// TwinCAT 3 PLC project convey
// ProgramVersion: 3.1.0.9
// libraries:
//   VisuElem3DPath, 3.5.6.0 (System)
//   VisuElemMeter, 3.5.6.0 (System)
//   VisuElems, 3.5.6.10 (System)
//   VisuElemsDateTime, 3.5.6.0 (System)
//   VisuElemsSpecialControls, 3.5.6.0 (System)
//   VisuElemsWinControls, 3.5.6.0 (System)
//   VisuElemTextEditor, 3.5.6.0 (System)
//   visuinputs, 3.5.6.0 (system)
//   VisuNativeControl, 3.5.6.0 (System)
//   Tc2_Standard, * (Beckhoff Automation GmbH)
//   Tc2_System, * (Beckhoff Automation GmbH)
//   Tc3_Interfaces, * (Beckhoff Automation GmbH)
//   Tc3_Module, * (Beckhoff Automation GmbH)
//   VisuDialogs, * (System)
// project tree:
//   / Buttons.TcIPO (not stored), GlobalImagePool.TcGIPO (not stored), GlobalTextList.TcGTLO, ImagePool.TcIPO (not stored), PlcTask.TcTTO, stateImages.TcIPO (not stored), Visualization Manager.TcVMO (not stored), VISU_TASK.TcTTO
//   GVLs/ GVL.TcGVL
//   POUs/ autoMode.TcPOU, caseImageUpdate.TcPOU, leftBelt.TcPOU, leftLift.TcPOU, MAIN.TcPOU, manualMode.TcPOU, bottomBelt.TcPOU, readState.TcPOU, relaxPistons.TcPOU, rightBelt.TcPOU, rightLift.TcPOU, topBelt.TcPOU
//   VISUs/ about.TcVIS, allControls.TcVIS, autoMode.TcVIS, Main.TcVIS, manualMode.TcVIS
// real-time tasks:
//   TASK PlcTask: cycle T#10ms, priority 20, ADS port 350
//   TASK VISU_TASK: cycle T#100000us, priority 30, ADS port 351
// I/O:
//   DEVICE Device 1 (EtherCAT), AmsNetId 172.24.66.56.2.1
//     Term 1 (EK1100) [EK1100 EtherCAT Coupler (2A E-Bus)]
//       Term 2 (EL1008) [EL1008 8Ch. Dig. Input 24V, 3ms]
//       Term 3 (EL2008) [EL2008 8Ch. Dig. Output 24V, 0.5A]
//       Term 4 (EL3002) [EL3002 2Ch. Ana. Input +/-10V]
//       Term 5 (EL4002) [EL4002 2Ch. Ana. Output 0-10V, 12bit]
//       Term 6 (EL3124) [EL3124 4Ch. Ana. Input 4-20mA Diff.]
//       Term 7 (EL4024) [EL4024 4Ch. Ana. Output 4-20mA, 12bit]
//       Term 10 (EL9011) [EL9011 End Terminal]
//     Term 8 (EK1100) [EK1100 EtherCAT Coupler (2A E-Bus)]
//       Box 9 (BK1250)
//   DEVICE Device 2 (EtherCAT Automation Protocol), AmsNetId 172.24.66.56.3.1
// variable links:
//   convey/convey Instance <-> Device 1 (EtherCAT)/Term 8 (EK1100)/Box 9 (BK1250)
//     PlcTask Inputs/GVL.I_bInput11 <-> Term 4 (KL1104)/Channel 3/GVL.I_bInput11
//     PlcTask Inputs/GVL.I_bInput12 <-> Term 4 (KL1104)/Channel 4/GVL.I_bInput12
//     PlcTask Inputs/GVL.I_bLeftLiftBottom <-> Term 3 (KL1104)/Channel 2/GVL.I_bLeftLiftBottom
//     PlcTask Inputs/GVL.I_bLeftLiftUp <-> Term 3 (KL1104)/Channel 1/GVL.I_bLeftLiftUp
//     PlcTask Inputs/GVL.I_bLowBeltLeft <-> Term 4 (KL1104)/Channel 1/GVL.I_bLowBeltLeft
//     PlcTask Inputs/GVL.I_bLowBeltRight <-> Term 3 (KL1104)/Channel 3/GVL.I_bLowBeltRight
//     PlcTask Inputs/GVL.I_bPieceLeftLift <-> Term 2 (KL1104)/Channel 1/GVL.I_bPieceLeftLift
//     PlcTask Inputs/GVL.I_bPieceRightLift <-> Term 2 (KL1104)/Channel 2/GVL.I_bPieceRightLift
//     PlcTask Inputs/GVL.I_bRightLiftBottom <-> Term 2 (KL1104)/Channel 4/GVL.I_bRightLiftBottom
//     PlcTask Inputs/GVL.I_bRightLiftUp <-> Term 2 (KL1104)/Channel 3/GVL.I_bRightLiftUp
//     PlcTask Inputs/GVL.I_bTopBeltRight <-> Term 3 (KL1104)/Channel 4/GVL.I_bTopBeltRight
//     PlcTask Inputs/GVL.I_bTopBeltleft <-> Term 4 (KL1104)/Channel 2/GVL.I_bTopBeltleft
//     PlcTask Outputs/GVL.O_bLeftLiftBeltLeft <-> Term 6 (KL2114)/Channel 4/GVL.O_bLeftLiftBeltLeft
//     PlcTask Outputs/GVL.O_bLeftLiftBeltRight <-> Term 6 (KL2114)/Channel 3/GVL.O_bLeftLiftBeltRight
//     PlcTask Outputs/GVL.O_bLeftLiftDown <-> Term 5 (KL2114)/Channel 2/GVL.O_bLeftLiftDown
//     PlcTask Outputs/GVL.O_bLeftLiftUp <-> Term 5 (KL2114)/Channel 1/GVL.O_bLeftLiftUp
//     PlcTask Outputs/GVL.O_bLowBeltLeft <-> Term 7 (KL2114)/Channel 4/GVL.O_bLowBeltLeft
//     PlcTask Outputs/GVL.O_bLowBeltRight <-> Term 7 (KL2114)/Channel 2/GVL.O_bLowBeltRight
//     PlcTask Outputs/GVL.O_bRightLiftBeltLeft <-> Term 6 (KL2114)/Channel 1/GVL.O_bRightLiftBeltLeft
//     PlcTask Outputs/GVL.O_bRightLiftBeltRight <-> Term 6 (KL2114)/Channel 2/GVL.O_bRightLiftBeltRight
//     PlcTask Outputs/GVL.O_bRightLiftDown <-> Term 5 (KL2114)/Channel 3/GVL.O_bRightLiftDown
//     PlcTask Outputs/GVL.O_bRightLiftUp <-> Term 5 (KL2114)/Channel 4/GVL.O_bRightLiftUp
//     PlcTask Outputs/GVL.O_bTopBeltLeft <-> Term 7 (KL2114)/Channel 1/GVL.O_bTopBeltLeft
//     PlcTask Outputs/GVL.O_bTopBeltRight <-> Term 7 (KL2114)/Channel 3/GVL.O_bTopBeltRight

CONFIGURATION convey
    RESOURCE PLC ON TwinCAT3
        TASK PlcTask(INTERVAL := T#10ms, PRIORITY := 20);
        TASK VISU_TASK(INTERVAL := T#100000us, PRIORITY := 30);
        PROGRAM MAIN WITH PlcTask : MAIN;
        PROGRAM VisuElems_Visu_Prg WITH VISU_TASK : VisuElems.Visu_Prg;
    END_RESOURCE
END_CONFIGURATION

// ---- GVLs/GVL.TcGVL
VAR_GLOBAL
	I_bPieceLeftLift              AT %I*: BOOL; // DI 1 - Piece in the left lift
	I_bPieceRightLift             AT %I*: BOOL; // DI 2 - Piece in the right lift
	I_bRightLiftBottom            AT %I*: BOOL; // DI 3 - Right lift is bottom
	I_bRightLiftUp                AT %I*: BOOL; // DI 4 - Right lift is up
	I_bLeftLiftBottom             AT %I*: BOOL; // DI 5 - Left lift is down
	I_bLeftLiftUp                 AT %I*: BOOL; // DI 6 - Left lift is up
	I_bLowBeltRight 	          AT %I*: BOOL; // DI 7 - Piece on low belt right side
	I_bTopBeltRight               AT %I*: BOOL; // DI 8 - Piece on top belt right side
	I_bLowBeltLeft                AT %I*: BOOL; // DI 9 - Piece on low belt left side
	I_bTopBeltleft                AT %I*: BOOL; // DI 10 - Piece on top belt left side
	I_bInput11                    AT %I*: BOOL; // DI 11 - Empty
	I_bInput12                    AT %I*: BOOL; // DI 12 - Empty
	I_STARTbutton				  AT %I*: BOOL;
	
	O_bLeftLiftUp                 AT %Q*: BOOL; // DO 1 - Left Lift up
	O_bLeftLiftDown               AT %Q*: BOOL; // DO 2 - Left Lift down
	O_bRightLiftDown              AT %Q*: BOOL; // DO 3 - Right Lift down
	O_bRightLiftUp                AT %Q*: BOOL; // DO 4 - Right Lift up
	O_bRightLiftBeltLeft          AT %Q*: BOOL; // DO 5 - Lift Right belt left
	O_bRightLiftBeltRight         AT %Q*: BOOL; // DO 6 - Lift Right belt right
	O_bLeftLiftBeltRight          AT %Q*: BOOL; // DO 7 - Lift Left belt right
	O_bLeftLiftBeltLeft           AT %Q*: BOOL; // DO 8 - Lift Left belt left
	O_bTopBeltLeft                AT %Q*: BOOL; // DO 9 - Top belt left
	O_bLowBeltRight               AT %Q*: BOOL; // DO 10 - Low belt right
	O_bTopBeltRight               AT %Q*: BOOL; // DO 11 - Top belt right
	O_bLowBeltLeft                AT %Q*: BOOL; // DO 12 - Low belt left
	Delay2:ton;
	state: INT;
END_VAR

// ---- POUs/MAIN.TcPOU
PROGRAM MAIN
VAR
	readState:readState;
	State: INT;
	autoMode: autoMode;
	relaxPistons:relaxPistons;
	manualMode:manualMode;
	stateVar: INT; 
	manualModeON:BOOL;
	autoModeON: BOOL;
	allControls: BOOL;
	bmpID: STRING;
	caseImageUpdate:caseImageUpdate;
	indusoftImage: STRING;
END_VAR

readState(caseState=>State);

	autoMode(ON:=autoModeON,caseState:=State);
	
	manualMode(ON:=manualModeON, toState:=stateVar, cState:=State, prevState=>);

relaxPistons();
caseImageUpdate(id:=State,bmpID=>bmpID,indusoftImage=>indusoftImage);

END_PROGRAM

// ---- POUs/readState.TcPOU
FUNCTION_BLOCK readState
VAR_INPUT
END_VAR
VAR_OUTPUT
	caseState : INT;
END_VAR
VAR
	counter : INT;
	value : LREAL;
	state : LREAL;
	inputArray: ARRAY[0..9] OF BOOL;
END_VAR

inputArray[0]:=I_bPieceLeftLift;
inputArray[1]:=I_bPieceRightLift;
inputArray[2]:=I_bRightLiftBottom;
inputArray[3]:=I_bRightLiftUp;
inputArray[4]:=I_bLeftLiftBottom;
inputArray[5]:=I_bLeftLiftUp;
inputArray[6]:=I_bLowBeltRight;
inputArray[7]:=I_bTopBeltRight;
inputArray[8]:=I_bLowBeltLeft;
inputArray[9]:=I_bTopBeltleft;

FOR counter :=0 TO 9 BY 1 DO
	IF inputArray[counter] THEN
		value := value + EXPT(2, counter);
	END_IF
END_FOR
state := value;
value := 0;
counter :=0;
caseState := LREAL_TO_INT(state);

END_FUNCTION_BLOCK

// ---- POUs/autoMode.TcPOU
FUNCTION_BLOCK autoMode
VAR_INPUT
	ON : BOOL;
	caseState : INT;
END_VAR
VAR_OUTPUT
END_VAR
VAR
	value : LREAL :=0;
	onDelay : TON;
	trigger : BOOL;
END_VAR

IF ON THEN
//AutoMode runtime :P
onDelay(IN:=I_bPieceLeftLift OR I_bPieceRightLift,pt:=T#2S,Q=>,ET=>);
//POSITION(1-8).LEFTLIFesRIGHTLIFT(0,1)
CASE caseState OF
	0: //do nothing
	21://1.0.1
	leftBelt(1);
	bottomBelt(1);
	topBelt(0);
	25: //1.0.0
	leftBelt(1);
	bottomBelt(1);
	topBelt(0);
	276://2.0.0 
	leftBelt(0);
	bottomBelt(1);
	280://2.0.1
	leftBelt(0);
	rightLift(4);
	bottomBelt(1);
	topBelt(0);
	292://2.1.0
	leftBelt(0);
	bottomBelt(1);
	topBelt(0);
	296://2.1.1
	leftBelt(0);
	rightLift(4);
	bottomBelt(1);
	topBelt(0);
	84://3.0.0
	rightBelt(1);
	bottomBelt(1);
	topBelt(0);
	88://3.0.1
	rightLift(4);
	rightBelt(1);
	bottomBelt(1);
	topBelt(0);
	100://3.1.0
	rightBelt(1);
	bottomBelt(1);
	topBelt(0);
	104://3.1.1
	rightLift(4);
	rightBelt(1);
	bottomBelt(1);
	topBelt(0);
	
	22://4.0.0
	IF onDelay.Q THEN
	rightbelt(0);
	bottomBelt(0);
	rightLift(3);
	END_IF
	38://4.1.0
	IF onDelay.Q THEN
	rightbelt(0);
	bottomBelt(0);
	rightLift(3);
	END_IF
	26://5.0.1
	rightBelt(2);
	topBelt(2);
	bottomBelt(0);
	42://5.1.1
	rightBelt(2);
	topBelt(2);
	bottomBelt(0);
	148://6.0.0
	leftLift(3);
	rightBelt(0);
	topBelt(2);
	bottomBelt(0);
	152://6.0.1
	leftLift(3);
	rightBelt(0);
	topBelt(2);
	bottomBelt(0);
	164://6.1.0
	rightBelt(0);
	topBelt(2);
	bottomBelt(0);
	168://6.1.1
	rightBelt(0);
	topBelt(2);
	bottomBelt(0);
	532://7.0.0
	leftLift(3);
	leftBelt(2);
	topBelt(2);
	bottomBelt(0);
	536://7.0.1
	leftLift(3);
	leftBelt(2);
	topBelt(2);
	bottomBelt(0);
	548://7.1.0
	leftBelt(2);
	topBelt(2);
	bottomBelt(0);
	552://7.1.1
	leftBelt(2);
	topBelt(2);
	bottomBelt(0);
	37://8.1.0
	IF onDelay.Q THEN
	leftBelt(0);
	topBelt(0);
	leftLift(4);
	END_IF
	41://8.1.1
	IF onDelay.Q THEN
	leftBelt(0);
	topBelt(0);
	leftLift(4);
	END_IF
END_CASE
END_IF
IF NOT ON AND NOT Main.allControls AND NOT MAIN.manualModeON THEN
	leftBelt(0);
	topBelt(0);
	rightBelt(0);
	bottomBelt(0);
END_IF

END_FUNCTION_BLOCK

// ---- POUs/leftBelt.TcPOU
FUNCTION leftBelt : BOOL
VAR_INPUT
	direction: INT :=0;
END_VAR
VAR
END_VAR

//The variable <direction> conventionaly can be initialized with the values:
//0 meaning STOP
//1 meaning RIGHT
//2 meaning LEFT
//3 meaning UP
//4 meaning DOWN
CASE direction OF
	0:
	O_bLeftLiftBeltLeft:=FALSE;
	O_bLeftLiftBeltRight :=FALSE;	
	1:
	O_bLeftLiftBeltLeft :=FALSE;
	O_bLeftLiftBeltRight :=TRUE;
	2:
	O_bLeftLiftBeltRight :=FALSE;
	O_bLeftLiftBeltLeft :=TRUE;
	
	ELSE
	O_bLeftLiftBeltLeft :=FALSE;
	O_bLeftLiftBeltRight :=FALSE;	
END_CASE

END_FUNCTION

// ---- POUs/bottomBelt.TcPOU
FUNCTION bottomBelt : BOOL
VAR_INPUT
	direction: INT :=0;
END_VAR
VAR
END_VAR

//The variable <direction> conventionaly can be initialized with the values:
//0 meaning STOP
//1 meaning RIGHT
//2 meaning LEFT
//3 meaning UP
//4 meaning DOWN
CASE direction OF
	0:
	O_bLowBeltLeft:=FALSE;
	O_bLowBeltRight:=FALSE;	
	1:
	O_bLowBeltLeft:=FALSE;
	O_bLowBeltRight:=TRUE;
	2:
	O_bLowBeltRight:=FALSE;
	O_bLowBeltLeft:=TRUE;
	
	ELSE
	O_bLowBeltLeft:=FALSE;
	O_bLowBeltRight:=FALSE;	
END_CASE

END_FUNCTION

// ---- POUs/topBelt.TcPOU
FUNCTION topBelt : BOOL
VAR_INPUT
	direction: INT := 0;
END_VAR
VAR
END_VAR

//The variable <direction> conventionaly can be initialized with the values:
//0 meaning STOP
//1 meaning RIGHT
//2 meaning LEFT
//3 meaning UP
//4 meaning DOWN
CASE direction OF
	0:
	O_bTopBeltLeft:=FALSE;
	O_bTopBeltRight:=FALSE;	
	1:
	O_bTopBeltLeft:=FALSE;
	O_bTopBeltRight:=TRUE;
	2:
	O_bTopBeltRight:=FALSE;
	O_bTopBeltLeft:=TRUE;
	
	ELSE
	O_bTopBeltLeft:=FALSE;
	O_bTopBeltRight:=FALSE;	
END_CASE

END_FUNCTION

// ---- POUs/rightLift.TcPOU
FUNCTION rightLift : BOOL
VAR_INPUT
	direction : INT :=0;
END_VAR
VAR
	//onDelay : TON;
END_VAR

//The variable <direction> conventionaly can be initialized with the values:
//0 meaning STOP
//1 meaning RIGHT
//2 meaning LEFT
//3 meaning UP
//4 meaning DOWN
CASE direction OF
	0:
	O_bRightLiftUp:=FALSE;
	O_bRightLiftDown:=FALSE;	
	3:
	O_bRightLiftDown:=FALSE;
	O_bRightLiftUp:=TRUE;
	//onDelay(IN:=TRUE,PT=T#2S,Q=>O_bRightLiftUp,ET=>);
	4:
	O_bRightLiftUp:=FALSE;
	O_bRightLiftDown:=TRUE;
	//onDelay(IN:=TRUE,PT=T#2S,Q=>O_bRightLiftDown,ET=>);	
	
	ELSE
	O_bLeftLiftUp:=FALSE;
	O_bLeftLiftDown:=FALSE;	
END_CASE

END_FUNCTION

// ---- POUs/rightBelt.TcPOU
FUNCTION rightBelt : BOOL

VAR_INPUT
	direction: INT :=0;
END_VAR
VAR
END_VAR

//The variable <direction> conventionaly can be initialized with the values:
//0 meaning STOP
//1 meaning RIGHT
//2 meaning LEFT
//3 meaning UP
//4 meaning DOWN
CASE direction OF
	0:
	O_bRightLiftBeltLeft:=FALSE;
	O_bRightLiftBeltRight :=FALSE;	
	1:
	O_bRightLiftBeltLeft :=FALSE;
	O_bRightLiftBeltRight :=TRUE;
	2:
	O_bRightLiftBeltRight :=FALSE;
	O_bRightLiftBeltLeft :=TRUE;
	
	ELSE
	O_bRightLiftBeltLeft :=FALSE;
	O_bRightLiftBeltRight :=FALSE;	
END_CASE

END_FUNCTION

// ---- POUs/leftLift.TcPOU
FUNCTION leftLift : BOOL
VAR_INPUT
	direction : INT :=0;
END_VAR
VAR
END_VAR

//The variable <direction> conventionaly can be initialized with the values:
//0 meaning STOP
//1 meaning RIGHT
//2 meaning LEFT
//3 meaning UP
//4 meaning DOWN
CASE direction OF
	0:
	O_bLeftLiftUp:=FALSE;
	O_bLeftLiftDown:=FALSE;	
	3:
	O_bLeftLiftDown:=FALSE;	
	O_bLeftLiftUp:=TRUE;
	4:
	O_bLeftLiftUp:=FALSE;	
	O_bLeftLiftDown:=TRUE;	
	//onDelay(IN:=TRUE,PT:=T#2S, Q=>O_bLeftLiftDown,ET=>);
	
	ELSE
	O_bLeftLiftUp:=FALSE;
	O_bLeftLiftDown:=FALSE;
END_CASE

END_FUNCTION

// ---- POUs/relaxPistons.TcPOU
FUNCTION_BLOCK relaxPistons
VAR_INPUT
END_VAR
VAR_OUTPUT
END_VAR
VAR
END_VAR

IF I_bRightLiftBottom THEN
	O_bRightLiftDown:=FALSE;
END_IF

IF  I_bRightLiftUp THEN
	O_bRightLiftUp:=FALSE;
END_IF

IF I_bLeftLiftBottom THEN
	O_bLeftLiftDown:=FALSE;
END_IF

IF  I_bLeftLiftUp THEN
	O_bLeftLiftUp:=FALSE;
END_IF

END_FUNCTION_BLOCK

// ---- POUs/manualMode.TcPOU
FUNCTION_BLOCK manualMode
VAR_INPUT
	ON : BOOL;
	toState: INT;
	cState: INT;
END_VAR
VAR_OUTPUT
	prevState : INT := 1;
END_VAR
VAR
	onDelay : TON;
END_VAR

IF ON THEN

CASE toState OF
	1:
	IF prevState = 2 THEN
		topBelt(2);
		leftBelt(2);
		leftLift(3);
	END_IF
	
	IF prevState = 8 THEN
		leftLift(3);
	END_IF
		prevState := 1;	
		
	2:
	IF prevState = 1 THEN
		topBelt(1);
		leftBelt(1);
	END_IF
	
	IF prevState = 3 THEN
		topBelt(2);
	END_IF
	prevState := 2;
	
	3:
	IF prevState = 2 THEN
		topBelt(1);
	END_IF
	
	IF prevState = 4 THEN
		topBelt(2);
		rightBelt(2);
	END_IF
	prevState := 3;
	
	4:
	IF prevState = 3 THEN
		topBelt(1);
		rightBelt(1);
		rightLift(3);
	END_IF
	
	IF prevState = 5 THEN
		rightLift(3);
	END_IF
	prevState := 4;
	
	5:
	IF prevState = 4 THEN
		rightLift(4);
	END_IF
	
	IF prevState = 6 THEN
		bottomBelt(1);
		rightBelt(1);
		rightLift(4);
	END_IF
	prevState := 5;
	
	6:
	IF prevState = 5 THEN
		bottomBelt(2);
		rightBelt(2);
	END_IF
	
	IF prevState = 7 THEN
		bottomBelt (1);
	END_IF
	prevState := 6;
	
	7:
	IF prevState = 6 THEN
		bottomBelt(2);
	END_IF
	
	IF prevState = 8 THEN
		bottomBelt(1);
		leftBelt(1);
	END_IF
	prevState := 7;
	
	8:
	IF prevState = 1 THEN
		leftLift(4);
	END_IF
	
	IF prevState = 7 THEN
		bottomBelt(2);
		leftBelt(2);
		leftLift(4);
	END_IF
	prevState := 8;
	
END_CASE

IF toState=2 AND (cState=552 OR cState=536 OR cState=532 OR cState=548) THEN
	topBelt(0);
	leftBelt(0);
END_IF

IF toState=3 AND (cState=168 OR cState=152 OR cState=148 OR cState=164) THEN
	topBelt(0);
	rightBelt(0);
END_IF

IF toState=6 AND (cState=104 OR cState=88 OR cState=84 OR cState=100) THEN
	bottomBelt(0);
	rightBelt(0);
END_IF

IF toState=7 AND (cState=296 OR cState=292 OR cState=276 OR cState=280) THEN
	bottomBelt(0);
	leftBelt(0);
END_IF

onDelay(IN:=(toState = 1 AND (cState = 41 OR cState=37)) OR (toState = 4 AND (cState = 42 OR cState=26)) OR (toState = 5 AND (cState = 38 OR cState=22)) OR (toState = 8 AND (cState = 21 OR cState=25)),PT:=T#2S,Q=>,ET=>);
//onDelay(IN:=toState = 2 AND (cState = 42 OR cState=26),PT:=T#2S,Q=>,ET=>);
//onDelay(IN:=toState = 5 AND (cState = 38 OR cState=22),PT:=T#2S,Q=>,ET=>);
//onDelay(IN:=toState = 8 AND (cState = 21 OR cState=25),PT:=T#2S,Q=>,ET=>);
IF onDelay.Q THEN
	bottomBelt(0);
	topBelt(0);
	rightBelt(0);
	leftBelt(0);
END_IF

END_IF

END_FUNCTION_BLOCK

// ---- POUs/caseImageUpdate.TcPOU
FUNCTION_BLOCK caseImageUpdate
VAR_INPUT
	id:INT;
END_VAR
VAR_OUTPUT
	bmpId:STRING;
	manualStateId:INT;
	indusoftImage:STRING;
END_VAR
VAR
	btn1:BOOL;
	btn2:BOOL;
	btn3:BOOL;
	btn4:BOOL;
	btn5:BOOL;
	btn6:BOOL;
	btn7:BOOL;
	btn8:BOOL;
	
END_VAR

IF id = 21 OR id =22 OR id = 24 OR id = 25 OR id = 26 OR id = 37 OR id = 38 OR id = 41 OR id = 42 OR id = 84 OR id = 88 OR id = 100 OR id = 104 OR id = 148 OR id = 164 OR id=168 OR id = 276 OR id = 280 OR id = 292 OR id = 296 OR id = 532 OR id = 536 OR id = 548 OR id = 552 THEN
	bmpId:=concat('stateImages.',INT_TO_STRING(id));
	indusoftImage:=concat(INT_TO_STRING(id), '.jpg');
	manualStateId:=id;

CASE id OF
	37, 41:
	btn1:=TRUE;
	btn2:=FALSE;
	btn3:=TRUE;
	btn4:=TRUE;
	btn5:=TRUE;
	btn6:=TRUE;
	btn7:=FALSE;
	btn8:=TRUE;
	532, 536, 548, 552:
	btn1:=FALSE;
	btn2:=FALSE;
	btn3:=TRUE;
	btn4:=TRUE;
	btn5:=TRUE;
	btn6:=TRUE;
	btn7:=TRUE;
	btn8:=TRUE;
	168, 164, 148, 24:
	btn1:=FALSE;
	btn2:=FALSE;
	btn3:=TRUE;
	btn4:=TRUE;
	btn5:=TRUE;
	btn6:=TRUE;
	btn7:=TRUE;
	btn8:=TRUE;
	26, 42:
	btn1:=FALSE;
	btn2:=TRUE;
	btn3:=TRUE;
	btn4:=FALSE;
	btn5:=TRUE;
	btn6:=TRUE;
	btn7:=TRUE;
	btn8:=TRUE; 
	22, 38:
	btn1:=TRUE;
	btn2:=TRUE;
	btn3:=FALSE;
	btn4:=TRUE;
	btn5:=TRUE;
	btn6:=FALSE;
	btn7:=TRUE;
	btn8:=TRUE;
	84, 88, 100, 104:
	btn1:=TRUE;
	btn2:=TRUE;
	btn3:=TRUE;
	btn4:=TRUE;
	btn5:=FALSE;
	btn6:=FALSE;
	btn7:=TRUE;
	btn8:=TRUE;
	276, 280, 292, 296:
	btn1:=TRUE;
	btn2:=TRUE;
	btn3:=TRUE;
	btn4:=TRUE;
	btn5:=FALSE;
	btn6:=FALSE;
	btn7:=TRUE;
	btn8:=TRUE;
	25, 21:
	btn1:=TRUE;
	btn2:=TRUE;
	btn3:=TRUE;
	btn4:=TRUE;
	btn5:=FALSE;
	btn6:=TRUE;
	btn7:=TRUE;
	btn8:=FALSE;
	
	
END_CASE
END_IF

END_FUNCTION_BLOCK

// ---- GlobalTextList.TcGTLO
TEXTLIST GlobalTextList
  32 = '"%d", state'
  34 = '%d'
  36 = '<'
  35 = '>'
  3 = 'auto control'
  5 = 'Auto control'
  33 = 'autoMode.state'
  13 = 'Back'
  15 = 'Belt'
  24 = 'Belt left'
  25 = 'Belt right'
  37 = 'DN'
  1 = 'GROUP 7'
  0 = 'GROUP NAME'
  10 = 'HAMEED QUREEB'
  9 = 'Ilir M Kokollari'
  11 = 'ILIR M KOKOLLARI'
  14 = 'Left lift'
  31 = 'Left lift Menu'
  27 = 'Lift down'
  29 = 'Lift left'
  30 = 'Lift right'
  26 = 'Lift up'
  18 = 'Low Belt'
  21 = 'Low left'
  23 = 'Low right'
  2 = 'Mannual control'
  12 = 'Manual control'
  4 = 'Quit'
  16 = 'Right lift'
  28 = 'Right lift Menu'
  6 = 'TOBILOBA ERO'
  17 = 'Top Belt'
  19 = 'Top left'
  20 = 'Top Right'
  22 = 'Top right'
  38 = 'UP'
  8 = 'WILPPU AHONEN'
  7 = 'ZHILUN CHANG'
  39 = '|'
END_TEXTLIST

// ---- VISUs/about.TcVIS
VISUALIZATION about  // 800x480
END_VISUALIZATION

// ---- VISUs/allControls.TcVIS
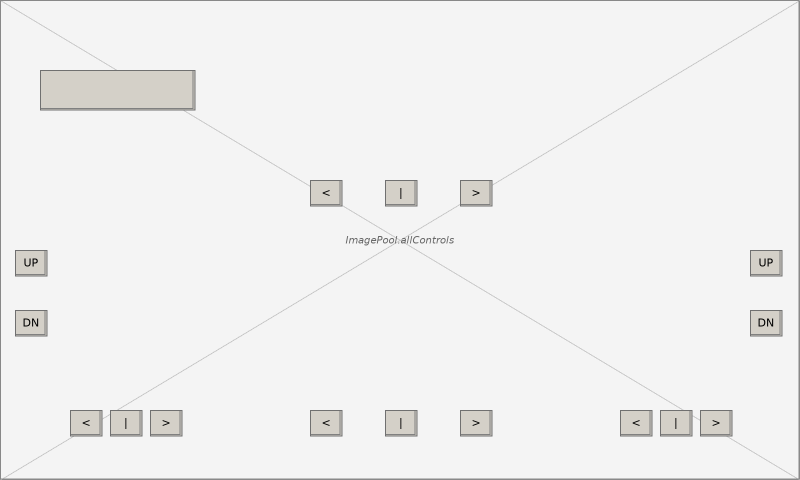
VISUALIZATION allControls  // 800x480
    Image (0,0 800x480), image: ImagePool.allControls
    Button (700,410 32x26), ">"
        OnMouseClick: execute { rightBelt(1); }
    Button (620,410 32x26), "<"
        OnMouseClick: execute { rightBelt(2); }
    Button (460,410 32x26), ">"
        OnMouseClick: execute { bottomBelt(1); }
    Button (310,410 32x26), "<"
        OnMouseClick: execute { bottomBelt(2); }
    Button (150,410 32x26), ">"
        OnMouseClick: execute { leftBelt(1); }
    Button (70,410 32x26), "<"
        OnMouseClick: execute { leftBelt(2); }
    Button (750,310 32x26), "DN"
        OnMouseClick: execute { rightLift(4); }
    Button (750,250 32x26), "UP"
        OnMouseClick: execute { rightLift(3); }
    Button (15,250 32x26), "UP"
        OnMouseClick: execute { leftLift(3); }
    Button (15,310 32x26), "DN"
        OnMouseClick: execute { leftLift(4); }
    Button (460,180 32x26), ">"
        OnMouseClick: execute { topBelt(1); }
    Button (310,180 32x26), "<"
        OnMouseClick: execute { topBelt(2); }
    Button (40,70 155x40), image: Buttons.homeButton
        OnMouseDown: change screen: Main
        OnMouseDown: execute { MAIN.allControls:=FALSE; }
    Button (110,410 32x26), "|"
        OnMouseClick: execute { leftBelt(0); }
    Button (385,410 32x26), "|"
        OnMouseClick: execute { bottomBelt(0); }
    Button (660,410 32x26), "|"
        OnMouseClick: execute { rightBelt(0); }
    Button (385,180 32x26), "|"
        OnMouseClick: execute { topBelt(0); }
END_VISUALIZATION

// ---- VISUs/autoMode.TcVIS
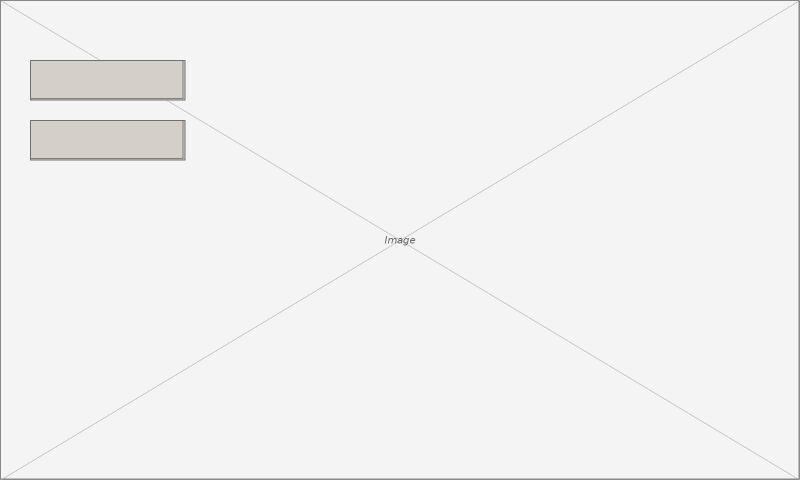
VISUALIZATION autoMode  // 800x480
    Image (0,0 800x480)
        p84334746: MAIN.bmpID
    Button (30,60 155x40), image: Buttons.homeButton
        OnMouseDown: change screen: Main
        OnMouseDown: execute { MAIN.autoModeON:=FALSE; }
    Button (30,120 155x40), image: Buttons.startButton
        OnMouseDown: toggle MAIN.autoModeON
END_VISUALIZATION

// ---- VISUs/Main.TcVIS
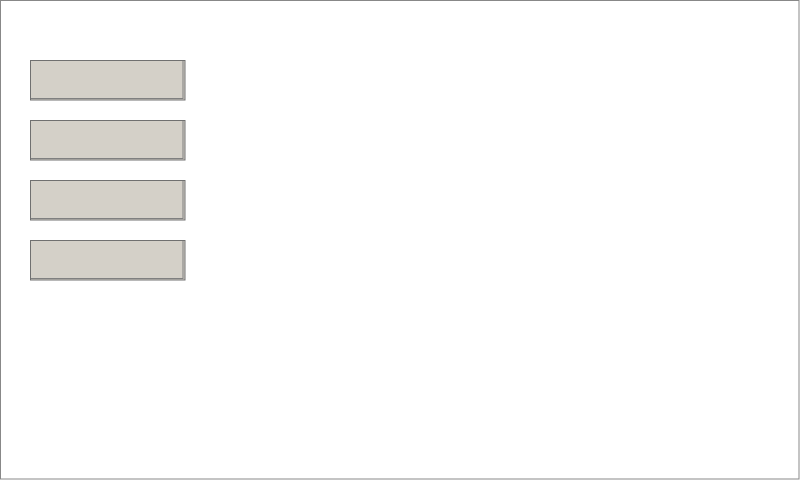
VISUALIZATION Main  // 800x480, background image ImagePool.homeScreen
    Button (30,60 155x40), image: Buttons.manualButton
        OnMouseClick: change screen: manualMode
    Button (30,120 155x40), image: Buttons.automaticButton
        OnMouseDown: change screen: autoMode
    Button (30,180 155x40), image: Buttons.controlButton
        OnMouseClick: change screen: allControls
        OnMouseClick: execute { MAIN.allControls:=TRUE; }
    Button (30,240 155x40), image: Buttons.aboutButton
        OnMouseClick: change screen: about
END_VISUALIZATION

// ---- VISUs/manualMode.TcVIS
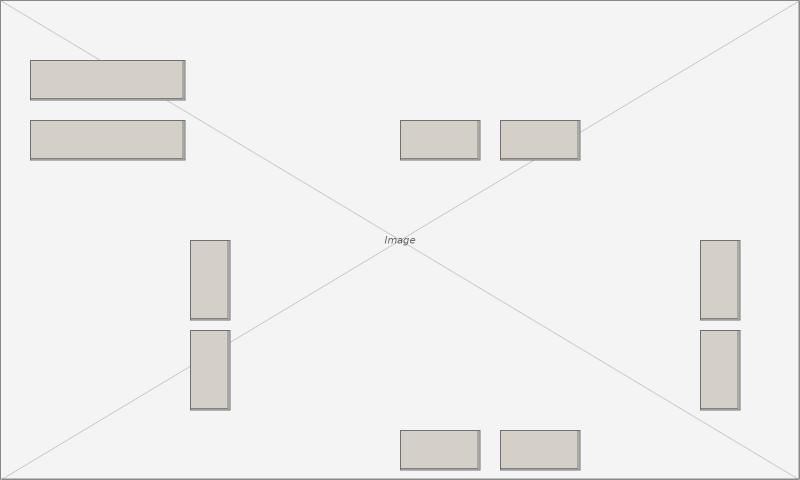
VISUALIZATION manualMode  // 800x480
    Image (0,0 800x480)
        p84334746: MAIN.bmpID
    Button (30,60 155x40), image: Buttons.homeButton
        OnMouseDown: change screen: Main
        OnMouseDown: execute { MAIN.manualModeON:=FALSE; }
    Button (30,120 155x40), image: Buttons.startButton
        OnMouseDown: toggle MAIN.manualModeON
    Button (190,330 40x80), invisible if: MAIN.caseImageUpdate.btn7, input disabled if: MAIN.caseImageUpdate.btn8, image: Buttons.down
        OnMouseClick: execute { Main.stateVar := 8; }
    Button (190,240 40x80), invisible if: MAIN.caseImageUpdate.btn8, input disabled if: MAIN.caseImageUpdate.btn8, image: Buttons.up
        OnMouseClick: execute { Main.stateVar := 1; }
    Button (700,240 40x80), invisible if: MAIN.caseImageUpdate.btn3, input disabled if: MAIN.caseImageUpdate.btn3, image: Buttons.up
        OnMouseClick: execute { Main.stateVar := 4; }
    Button (700,330 40x80), invisible if: MAIN.caseImageUpdate.btn4, input disabled if: MAIN.caseImageUpdate.btn4, image: Buttons.down
        OnMouseClick: execute { Main.stateVar := 5; }
    Button (500,430 80x40), invisible if: MAIN.caseImageUpdate.btn5, input disabled if: MAIN.caseImageUpdate.btn5, image: Buttons.right
        OnMouseClick: execute {
            IF MAIN.manualMode.prevState = 8 THEN
            	Main.stateVar := 7;
            END_IF
            IF MAIN.manualMode.prevState = 7 THEN
            	Main.stateVar := 6;
            END_IF
            IF MAIN.manualMode.prevState = 6 THEN
            	Main.stateVar := 5;
            END_IF
        }
    Button (400,430 80x40), invisible if: MAIN.caseImageUpdate.btn6, input disabled if: MAIN.caseImageUpdate.btn6, image: Buttons.left
        OnMouseClick: execute {
            IF MAIN.manualMode.prevState = 5 THEN
            	Main.stateVar := 6;
            END_IF
            IF MAIN.manualMode.prevState = 6 THEN
            	Main.stateVar := 7;
            END_IF
            IF MAIN.manualMode.prevState = 7 THEN
            	Main.stateVar := 8;
            END_IF
        }
    Button (400,120 80x40), invisible if: MAIN.caseImageUpdate.btn1, input disabled if: MAIN.caseImageUpdate.btn1, image: Buttons.left
        OnMouseClick: execute {
            IF MAIN.manualMode.prevState = 2 THEN
            	Main.stateVar := 1;
            END_IF
            IF MAIN.manualMode.prevState = 3 THEN
            	Main.stateVar := 2;
            END_IF
            IF MAIN.manualMode.prevState = 4 THEN
            	Main.stateVar := 3;
            END_IF
        }
    Button (500,120 80x40), invisible if: MAIN.caseImageUpdate.btn2, input disabled if: MAIN.caseImageUpdate.btn2, image: Buttons.right
        OnMouseClick: execute {
            IF MAIN.manualMode.prevState = 1 THEN
            	Main.stateVar := 2;
            END_IF
            IF MAIN.manualMode.prevState = 2 THEN
            	Main.stateVar := 3;
            END_IF
            IF MAIN.manualMode.prevState = 3 THEN
            	Main.stateVar := 4;
            END_IF
        }
END_VISUALIZATION
